PROGRAM PRG_DET_SLIT
VAR
	fbSlits_Det: FB_Slits;
	bExecuteMotion: BOOL := TRUE;
	bMoveOk: BOOL :=TRUE;
	bInit:BOOL:=TRUE;
END_VAR

// 4 jaws slit

IF bInit THEN
	bInit := FALSE;
	
	GVL_Main.M18.nBrakeMode := ENUM_StageBrakeMode.NO_BRAKE;
	GVL_Main.M18.bHardwareEnable := TRUE;
	GVL_Main.M18.bPowerSelf := TRUE;
	
	GVL_Main.M19.nBrakeMode := ENUM_StageBrakeMode.NO_BRAKE;
	GVL_Main.M19.bHardwareEnable := TRUE;
	GVL_Main.M19.bPowerSelf := TRUE;
	GVL_Main.M20.nBrakeMode := ENUM_StageBrakeMode.NO_BRAKE;
	GVL_Main.M20.bHardwareEnable := TRUE;
	GVL_Main.M20.bPowerSelf := TRUE;
	GVL_Main.M21.nBrakeMode := ENUM_StageBrakeMode.NO_BRAKE;
	GVL_Main.M21.bHardwareEnable := TRUE;
	GVL_Main.M21.bPowerSelf := TRUE;
	
	
	//
	GVL_Main.M18.nEnableMode := ENUM_StageEnableMode.DURING_MOTION ;
	GVL_Main.M19.nEnableMode := ENUM_StageEnableMode.DURING_MOTION ;
	GVL_Main.M20.nEnableMode := ENUM_StageEnableMode.DURING_MOTION ;
	GVL_Main.M21.nEnableMode := ENUM_StageEnableMode.DURING_MOTION ;
END_IF
fbSlits_Det(	i_DevName:=					'DET_SLITS',
				stTopBlade:=				GVL_Main.M20,
				stBottomBlade:=				GVL_Main.M21,
				stLeftBlade:=				GVL_Main.M18,
				stRightBlade:=				GVL_Main.M19,
				io_fbFFHWO:=				GVL_PMPS.io_fbFFHWO,
				fbArbiter:=					GVL_PMPS.fbArbiter,
				bExecuteMotion:=			bExecuteMotion,
				bMoveOk:=					bMoveOk
);

END_PROGRAM

(* stored: Version 1.1.0.1, ProductVersion 3.1.4022.18
   POU PRG_DET_SLIT: Id {2eb18d0f-2877-4c70-a778-30d760427220}, SpecialFunc None *)
